FUNCTION_BLOCK FB_Counter
VAR
END_VAR

METHOD GetSignedDelta : UDINT
VAR_INPUT
    a : INT;
    b : INT;
END_VAR
GetSignedDelta := DINT_TO_UDINT(INT_TO_DINT(a) - INT_TO_DINT(b));
END_METHOD

END_FUNCTION_BLOCK

(* stored: Version 1.1.0.1
   POU FB_Counter: Id {3086daba-f4bd-45e6-88ad-83c11b2184d2}, SpecialFunc None
   Method GetSignedDelta: Id {a36f162b-75c1-4b02-9372-bbdbeb9b6b67} *)
